// Block: PPrgArchive6

DATA_BLOCK PPrgArchive6
VERSION : 0.1
   NON_RETAIN
   VAR
      PRG : Array[501..600] of PPrg_Data;
   END_VAR

BEGIN
   // No initialization required
END_DATA_BLOCK
